{attribute 'reflection'}
FUNCTION_BLOCK T_AssertionListenerMock IMPLEMENTS I_AssertionListener
VAR
    {attribute 'instance-path'} 
    {attribute 'no_init'}
    _FullTestName : T_MaxString; // Automatically initialised with the full name of the instance
    _TestName : T_MaxString; 
    _AssertionFailed  : BOOL;
    _AssertionMessage : T_MaxString;
    _ExpectedAsString : T_MaxString;
    _ActualAsString   : T_MaxString;
END_VAR

PROPERTY ActualAsString : T_MaxString
GET
ActualAsString := _ActualAsString;
END_GET
SET
_ActualAsString := ActualAsString;
END_SET
END_PROPERTY

PROPERTY AssertionFailed : BOOL
GET
AssertionFailed := _AssertionFailed;
END_GET
SET
_AssertionFailed := AssertionFailed;
END_SET
END_PROPERTY

PROPERTY AssertionMessage : T_MaxString
GET
AssertionMessage := _AssertionMessage;
END_GET
SET
_AssertionMessage := AssertionMessage;
END_SET
END_PROPERTY

PROPERTY ExpectedAsString : T_MaxString
GET
ExpectedAsString := _ExpectedAsString;
END_GET
SET
_ExpectedAsString := ExpectedAsString;
END_SET
END_PROPERTY

METHOD OnAssertionFailed
VAR_INPUT
    AssertionMessage : T_MaxString;
    ExpectedAsString : T_MaxString;
    ActualAsString   : T_MaxString;
END_VAR
_AssertionFailed   := TRUE;
_AssertionMessage  := AssertionMessage;
_ExpectedAsString := ExpectedAsString;
_ActualAsString := ActualAsString;
END_METHOD

PROPERTY TestName : Tc2_System.T_MaxString
GET
VAR_INST
    StringSplitter : T_StringSplitter;
END_VAR
IF _TestName = '' THEN
   
    StringSplitter.Init(
        Str := _FullTestName,
        Delim1 := '.',
        Delim2 := '');
    
    WHILE StringSplitter.HasMore() DO
        _TestName := StringSplitter.GetNext(); // to get last sub-section
    END_WHILE
   
END_IF

TestName := _TestName;
END_GET
END_PROPERTY

END_FUNCTION_BLOCK

(* stored: Version 1.1.0.1, ProductVersion 3.1.4024.4
   POU T_AssertionListenerMock: Id {aea5748a-7a0b-49d1-9b5d-092bdfc42755}, SpecialFunc None
   Folder Methods: Id {c58fa9bc-ee0f-4be9-9454-767cd276a46b}
   Folder Properties: Id {04e2c3c7-c554-4932-b678-dc45a6ac1436}
   Property ActualAsString: Id {cfa9e900-1b4f-4c58-88f7-0c37474fc2cf}
   Get Get: Id {67be1d0c-f2d6-49b4-aeb6-695ff5eef1d9}
   Set Set: Id {fd8da95b-1746-4f44-95bb-f29cdb43f6fa}
   Property AssertionFailed: Id {e844e423-5b4f-4e3c-a75d-c5915f5ba038}
   Get Get: Id {55a92eae-047c-4cca-ad3e-e52d8ff147bf}
   Set Set: Id {ec0aec31-1391-4218-b50b-da4c10c6f7f5}
   Property AssertionMessage: Id {37f7cb1e-4125-4635-8207-039575e7a88f}
   Get Get: Id {b835a9e1-6698-4fd3-966b-d2e0544064fc}
   Set Set: Id {f096403a-15cd-4d8c-9be9-d40130c76db9}
   Property ExpectedAsString: Id {aefafe6d-e23e-44d0-b665-c75fbe1b7e6e}
   Get Get: Id {bf0c3a84-0f42-45be-80d8-115af0271dc7}
   Set Set: Id {86bef8f9-6aba-496a-9310-da84fce1ffdc}
   Method OnAssertionFailed: Id {a572523e-eb6e-4cc0-a62e-e3d15590ca01}
   Property TestName: Id {0835bb46-063f-406a-a937-e9d212ba8cbf}
   Get Get: Id {af1bd727-18ac-4d78-9390-07553b1c082b} *)
